Staubli VAL3: recvHeartbeat.pgx

public program recvHeartbeat()
  local num l_nByte
  local num l_nBytesRecv
  local num l_nHtbt
  local num l_nHtbtB[4]
  local num l_nIndex
begin
  // Copyright (c) 2016, Ocado Technology - Robotics Research Team
  //
  // Licensed under the Apache License, Version 2.0 (the "License");
  // you may not use this file except in compliance with the License.
  // You may obtain a copy of the License at
  //
  //     http://www.apache.org/licenses/LICENSE-2.0
  //
  // Unless required by applicable law or agreed to in writing, software
  // distributed under the License is distributed on an "AS IS" BASIS,
  // WITHOUT WARRANTIES OR CONDITIONS OF ANY KIND, either express or implied.
  // See the License for the specific language governing permissions and
  // limitations under the License.



  while (true)
    l_nBytesRecv=0
    l_nIndex = sioGet(siTcpIpFbk, l_nByte)
    if (l_nIndex == -1)
      // connection not established or connection lost
      if (nOutConnFlag == 1)
        nOutConnFlag = -1
      endIf
    else
      // it means l_nIndex >= 0: connection established
      // check if connection had not already been established
      if (nOutConnFlag != 1)
        // delay data output to avoid sync issues with client
        delay(1.0)
        // flag connection as established
        nOutConnFlag = 1
      endIf
    endIf
  endWhile
end
